(* IEC 61131-3 sources: Industry-PLC-LLM/data/PLCBEAD_repo/PLCBEAD_PLCEmbed-main/PLC-BEAD/Source/GEB/FT_PID, 1 file *)

(* ---- FT_PID.ST ---- *)
FUNCTION_BLOCK T_PLC_US_Block
	VAR_OUTPUT
		T_PLC_US :	UDINT;
	END_VAR

	VAR
		PLC_TICKS_PER_SEC :	INT;
		PLC_SYS_TICK_CNT :	DINT;
	END_VAR

	VAR
		debug :	BOOL;
		N :	INT;
		Offset :	UDINT;
		temp :	DWORD := DWORD#1;
		MODE :	BOOL;
		faktor :	UDINT;
		init :	BOOL;
		v_plc_ticks_per_sec :	UDINT;
		base :	UDINT := UDINT#1000000;
	END_VAR

	IF init = FALSE THEN
		v_plc_ticks_per_sec := INT_TO_UDINT(PLC_TICKS_PER_SEC);
		IF v_plc_ticks_per_sec = UDINT#1024 THEN
			faktor := UDINT#1000;
			MODE := FALSE;
		ELSIF v_plc_ticks_per_sec > UDINT#0 THEN
			IF v_plc_ticks_per_sec <= base THEN
				faktor := base / v_plc_ticks_per_sec;
				MODE := FALSE;
			ELSE
				faktor := v_plc_ticks_per_sec / base;
				MODE := TRUE;
			END_IF;
		ELSE
			faktor := UDINT#1;
		END_IF;
		init := TRUE;
	END_IF;

	IF MODE THEN
		T_PLC_US := DINT_TO_UDINT(PLC_SYS_TICK_CNT) / faktor;
	ELSE
		T_PLC_US := DINT_TO_UDINT(PLC_SYS_TICK_CNT) * faktor;
	END_IF;

	IF debug THEN
		T_PLC_US := (DWORD_TO_UDINT(SHL(UDINT_TO_DWORD(T_PLC_US),N) OR SHL(temp,N)) - UDINT#1) + Offset;
	END_IF;
END_FUNCTION_BLOCK

FUNCTION_BLOCK T_PLC_MS_block
	VAR_OUTPUT
		T_PLC_MS :	UDINT;
	END_VAR

	VAR
		PLC_TICKS_PER_SEC :	INT;
		PLC_SYS_TICK_CNT :	DINT;
	END_VAR

	VAR
		debug :	BOOL;(*Debug-Mode ON / OFF*)
		N :	INT;(*Debug-Faktor*)
		Offset :	UDINT;(*Debug-Offset*)
		temp :	DWORD := DWORD#1;(*Debug-Offset*)
		MODE :	BOOL;(*modus*)
		faktor :	UDINT;(*Systemtakt-Faktor*)
		init :	BOOL;
		v_plc_ticks_per_sec :	UDINT;
		base :	UDINT := UDINT#1000;
	END_VAR

	IF init = FALSE THEN
		v_plc_ticks_per_sec := INT_TO_UDINT(PLC_TICKS_PER_SEC);
		IF v_plc_ticks_per_sec = UDINT#1024 THEN
			faktor := UDINT#1;
			MODE := FALSE;
		ELSIF v_plc_ticks_per_sec > UDINT#0 THEN
			IF v_plc_ticks_per_sec <= base THEN
				faktor := base / v_plc_ticks_per_sec;
				MODE := FALSE;
			ELSE
				faktor := v_plc_ticks_per_sec / base;
				MODE := TRUE;
			END_IF;
		ELSE
			faktor := UDINT#1;
		END_IF;
		init := TRUE;
	END_IF;

	IF MODE THEN
		T_PLC_MS := DINT_TO_UDINT(PLC_SYS_TICK_CNT) / faktor;
	ELSE
		T_PLC_MS := DINT_TO_UDINT(PLC_SYS_TICK_CNT) * faktor;
	END_IF;

	IF debug THEN
		T_PLC_MS := (DWORD_TO_UDINT(SHL(UDINT_TO_DWORD(T_PLC_MS),N) OR SHL(temp,N)) - UDINT#1) + Offset;
	END_IF;
END_FUNCTION_BLOCK

FUNCTION_BLOCK INTEGRATE

	VAR_INPUT
		E :	BOOL := TRUE;
		X :	REAL;
		K :	REAL := 1.0;
	END_VAR

	VAR_IN_OUT
		Y :	REAL;
	END_VAR

	VAR
		X_LAST :	REAL;
		init :	BOOL;
		T_PLC_MS :	T_PLC_MS_block;
		last :	UDINT;
		TX :	UDINT;
	END_VAR

	T_PLC_MS();
	TX:= T_PLC_MS.T_PLC_MS;

	IF NOT init THEN
		init := TRUE;
		X_LAST := X;
	ELSIF E THEN
		Y := (X + X_LAST) * 0.5E-3 * UDINT_TO_REAL(TX-last) * K + Y;
		X_LAST := X;
	END_IF;
	last := TX;

END_FUNCTION_BLOCK

FUNCTION_BLOCK FT_INT_Block

	VAR_INPUT
		IN :	REAL;
		K :	REAL := 1.0;
		RUN :	BOOL := TRUE;
		RST :	BOOL;
		OUT_MIN :	REAL := REAL#-1.0E-37;
		OUT_MAX :	REAL := REAL#1.0E37;
	END_VAR

	VAR_OUTPUT
		OUT :	REAL;
		LIM :	BOOL;
	END_VAR

	VAR
		INTEG :	INTEGRATE;
	END_VAR

	IF RST THEN
		OUT := 0.0;
	ELSE
		INTEG(X := IN, E := RUN, K := K, Y := OUT);
		OUT := INTEG.Y;
	END_IF;

	(* limit the OUTputs *)
	IF OUT >= OUT_MAX THEN
		OUT := OUT_MAX;
		LIM := TRUE;
	ELSIF OUT <= OUT_MIN THEN
		OUT := OUT_MIN;
		LIM := TRUE;
	ELSE
		LIM := FALSE;
	END_IF;

END_FUNCTION_BLOCK

FUNCTION_BLOCK FT_DERIV
	VAR_INPUT
		IN :	REAL;
		K :	REAL := 1.0;
		RUN :	BOOL := TRUE;
	END_VAR

	VAR_OUTPUT
		OUT :	REAL;
	END_VAR

	VAR
		old :	REAL;
		TX :	UDINT;
		last :	UDINT;
		init :	BOOL;
		tc :	REAL;
		T_PLC_US :	T_PLC_US_Block;
	END_VAR

	T_PLC_US();
	TX:= T_PLC_US.T_PLC_US;
	tc := UDINT_TO_REAL(TX - last);

	IF NOT init THEN
		init := TRUE;
		old := IN;
	ELSIF RUN AND tc > 0.0 THEN
		OUT := (IN - old) / tc * 1000000.0 * K;
		old := IN;
	ELSE
		OUT := 0.0;
	END_IF;

	last := TX;

	T_PLC_US();
	TX:= T_PLC_US.T_PLC_US;

	IF NOT init THEN
		init := TRUE;
	ELSIF RUN AND (TX - last) > UDINT#0 THEN
		OUT := (IN - old) / UDINT_TO_REAL(TX - last) * 1000000.0 * K;
	ELSE
		OUT := 0.0;
	END_IF;
	old := IN;
	last := TX;
END_FUNCTION_BLOCK

FUNCTION_BLOCK FT_PID

	VAR_INPUT
		IN :	REAL;
		KP :	REAL := 1.0;
		TN :	REAL := 1.0;
		TV :	REAL := 1.0;
		ILIM_L :	REAL := -1.0E38;
		ILIM_H :	REAL := 1.0E38;
		IEN :	BOOL := TRUE;
		RST :	BOOL := FALSE;
	END_VAR

	VAR_OUTPUT
		Y :	REAL;
		LIM :	BOOL;
	END_VAR

	VAR
		INTEG :	FT_INT_Block;
		diff :	FT_DERIV;
	END_VAR

	IF TN > 0.0 THEN
		INTEG(IN := IN, K := 1.0 / TN, RUN := IEN, RST := RST, OUT_MIN := ILIM_L, OUT_MAX := ILIM_H);
	ELSE
		INTEG(RST := FALSE);
	END_IF;

	(* run differentiator *)
	diff(IN := IN, K := TV);

	(* combine both VALues *)
	Y := KP * (INTEG.OUT + diff.OUT + IN);

	(* check if INTEGrator has reached its limits and set OVERFLOW *)
	LIM := INTEG.LIM;

END_FUNCTION_BLOCK

PROGRAM program0
	VAR
		IN :	REAL;
		KP :	REAL := 1.0;
		TN :	REAL := 1.0;
		TV :	REAL := 1.0;
		ILIM_L :	REAL := -1.0E38;
		ILIM_H :	REAL := 1.0E38;
		IEN :	BOOL := TRUE;
		RST :	BOOL := FALSE;

		Y :	REAL;
		LIM :	BOOL;

		func_block : FT_PID;
	END_VAR
	func_block.IN :=IN;
	func_block.KP :=KP;
	func_block.TN :=TN;
	func_block.TV :=TV;
	func_block.ILIM_L :=ILIM_L;
	func_block.ILIM_H :=ILIM_H;
	func_block.IEN :=IEN;
	func_block.RST :=RST;

	func_block();
	Y := func_block.Y;
	LIM := func_block.LIM;
END_PROGRAM
